// TIA Portal V19 export
TYPE "typePressureGuageRs485Interface"
TITLE = LBC_typeAnalogOutputInterface
// Module interface for external systems
// stored: Access Published
   STRUCT
      commands : "LBC_typeInterfaceCommands";
      monitoring : "typePressureGuageRs485AnalogProcessValues";
      configuration : "typePressureGuageRs485Configuration";
   END_STRUCT;
END_TYPE
